// TIA Portal V20 export
ORGANIZATION_BLOCK "Main"   // OB1016, LAD, ProgramCycle
TITLE = "Main Program Sweep (Cycle)"
// stored: AutoNumber false, IsIECCheckEnabled true, Namespace Unit1.Em2, SetENOAutomatically true
   VAR_INPUT
      Initial_Call : Bool;   // Initial call of this OB
      Remanence : Bool;   // =True, if remanent data are available
   END_VAR
   VAR_TEMP
      tempIndex : Int;   // Index of EM in the array
   END_VAR
BEGIN

REGION Network 1: Simulation
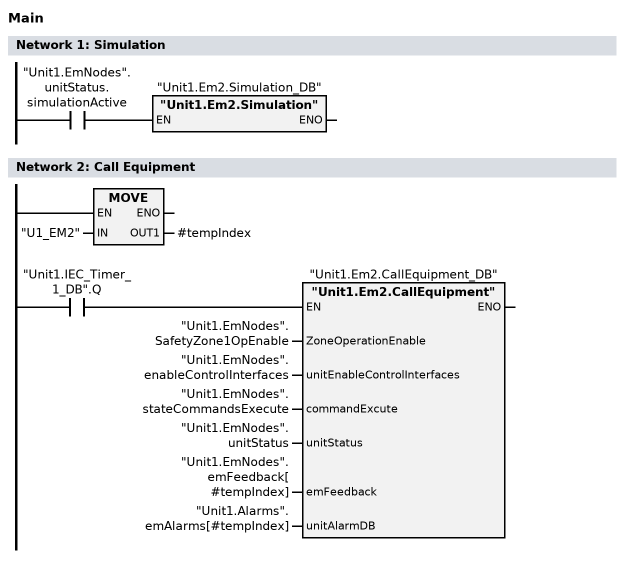
   RUNG wire#powerrail
      Contact( "Unit1.EmNodes".unitStatus.simulationActive )
      "Unit1.Em2.Simulation_DB"()
   END_RUNG
   // the same network as SCL:
   IF "Unit1.EmNodes".unitStatus.simulationActive THEN
       "Unit1.Em2.Simulation_DB"();   // "Unit1.Em2.Simulation"
   END_IF;
END_REGION

REGION Network 2: Call Equipment
   RUNG wire#powerrail
      Move(in := "U1_EM2", out1 => #tempIndex)
   END_RUNG
   RUNG wire#powerrail
      Contact( "Unit1.IEC_Timer_1_DB".Q )
      "Unit1.Em2.CallEquipment_DB"(ZoneOperationEnable := "Unit1.EmNodes".SafetyZone1OpEnable, unitEnableControlInterfaces := "Unit1.EmNodes".enableControlInterfaces, commandExcute := "Unit1.EmNodes".stateCommandsExecute, unitStatus := "Unit1.EmNodes".unitStatus, emFeedback := "Unit1.EmNodes".emFeedback[#tempIndex], unitAlarmDB := "Unit1.Alarms".emAlarms[#tempIndex])
   END_RUNG
   // the same network as SCL:
   #tempIndex := "U1_EM2";
   IF "Unit1.IEC_Timer_1_DB".Q THEN
       "Unit1.Em2.CallEquipment_DB"(ZoneOperationEnable := "Unit1.EmNodes".SafetyZone1OpEnable,   // "Unit1.Em2.CallEquipment"
                               unitEnableControlInterfaces := "Unit1.EmNodes".enableControlInterfaces,
                               commandExcute := "Unit1.EmNodes".stateCommandsExecute,
                               unitStatus := "Unit1.EmNodes".unitStatus,
                               emFeedback := "Unit1.EmNodes".emFeedback[#tempIndex],
                               unitAlarmDB := "Unit1.Alarms".emAlarms[#tempIndex]);
   END_IF;
END_REGION
END_ORGANIZATION_BLOCK
